TYPE ST_INPUTS_Unit_OzoneGenerator:
STRUCT
	
	Mode:     		E_DeviceMode;
	Command:     E_DeviceState;

END_STRUCT
END_TYPE

(* stored: Version 1.1.0.1, ProductVersion 3.1.4024.12
   DUT ST_INPUTS_Unit_OzoneGenerator: Id {9bc4289e-d115-430f-b79a-f51352bf496a} *)
